{attribute 'GeneratedUsingTerminal: EL6601--0000'}
{attribute addProperty BoxType "EL6601--0000"}
{attribute addProperty Id "InfoDataAT %I*InfoData_32EB74EA10"}
{attribute addProperty CRC "4004708084"}
{attribute addProperty Size "10"}
TYPE EL6601_EEB2FEF4 EXTENDS EtcSlaveTerminalBase_947E5A46 :
STRUCT
	{attribute addProperty Name "InfoData"}
	InfoData : InfoData_32EB74EA;
END_STRUCT
END_TYPE

(* stored: Version 1.2.0.0, ProductVersion 3.1.4024.9
   DUT EL6601_EEB2FEF4: Id {8b9c7b52-91d0-40ea-b61a-b613d65eaf27} *)
